FUNCTION_BLOCK FB_Sample_WidgetBase IMPLEMENTS I_Sample_WidgetInterface
VAR
    _sAdsPath : STRING(255);
    _sAttr1   : STRING(80);
    _nCalls   : UDINT;
END_VAR

;

METHOD BuildAttributes : UDINT
VAR_INPUT
    nFlags : DWORD;
END_VAR
_nCalls         := _nCalls + 1;
BuildAttributes := _nCalls;
END_METHOD

METHOD ProcessCommand : BOOL
VAR_INPUT
    nCommandId : DINT;
    fValue     : LREAL;
END_VAR
VAR_OUTPUT
    bHandled   : BOOL;
END_VAR
IF nCommandId = 1 THEN
    bHandled       := TRUE;
    ProcessCommand := TRUE;
ELSE
    bHandled       := FALSE;
    ProcessCommand := FALSE;
END_IF
END_METHOD

PROPERTY AdsPath : STRING(255)
GET
AdsPath := _sAdsPath;
END_GET
END_PROPERTY

PROPERTY AttributeVariable1 : STRING(80)
GET
AttributeVariable1 := _sAttr1;
END_GET
SET
_sAttr1 := AttributeVariable1;
END_SET
END_PROPERTY

END_FUNCTION_BLOCK

(* stored: Version 1.1.0.1, ProductVersion 3.1.4024.16
   POU FB_Sample_WidgetBase: Id {a3e34305-39bd-401e-826d-695855db68cd}, SpecialFunc None
   Method BuildAttributes: Id {aa5156df-01bb-4d37-922f-796bfdfe7723}
   Method ProcessCommand: Id {6dc72b73-e4a9-4566-a0d8-547e4e44192e}
   Property AdsPath: Id {f02b1906-9272-490d-9c35-9ea74e3ca803}
   Get Get: Id {2f2fa5e8-af38-42a5-a3a2-ed1338544c1a}
   Property AttributeVariable1: Id {3188c954-2131-4fa7-bb18-e4dad809d8c5}
   Get Get: Id {ef8501fa-ed4c-416a-8ffa-d9055c9e3ddc}
   Set Set: Id {1c780ff0-aa58-4e3d-98aa-7bef5cc9a12a} *)
